// TIA Portal V18 export
// export: Created 2026-06-11T07:10:00.0000000Z, ExportSetting WithDefaults, DisplayName Totally Integrated Automation Portal, DisplayVersion V18, DisplayName WinCC Professional, DisplayVersion V18
Screen "Screen_Login"  1920x1080, Number=2
  ScreenLayer 
    TextField "Text_field_3005" at 360,200 size 1200x80  Text="<body><p>HỆ THỐNG ĐIỀU KHIỂN VÀ GIÁM SÁT MIXING</p></body>"
    TextField "Text_field_300B" at 360,280 size 1200x40  Text="<body><p>DỰ ÁN LIÊN GIA BẢO - AREA 1400</p></body>"
    Rectangle "Panel_Login_Background" at 710,380 size 500x280
    Button "Btn_Screen_Login" at 760,420 size 400x50  TextOff="<body><p>ĐĂNG NHẬP (LOGIN)</p></body>"
      on Click: ShowLogonDialog()
    Button "Btn_Screen_Logout" at 760,490 size 400x50  TextOff="<body><p>ĐĂNG XUẤT (LOGOFF)</p></body>"
      on Click: Logoff()
    Button "Btn_Enter_System" at 760,560 size 400x50  TextOff="<body><p>VÀO HỆ THỐNG (ENTER SYSTEM)</p></body>"
      on Click: ActivateScreen(Screen name := Screen_1, Object number := 0)
